Staubli VAL3: readDET.pgx

program readDET()
  local num l_nError
  local string l_sValue
begin
  // Read current value from conveyor library
  resize(sCaption,1,pg:nNumOfTxtBox)
  call pg:getCaption(sCaption)
  call ut:_toString(det:nMaxNumOfObject,"",l_sValue)
  call pg:setFieldValue(sCaption[0],l_sValue,l_nError)
end
